FUNCTION_BLOCK FB_HMI_RP_BRANCH_A EXTENDS FB_HMI_COMPONENT
VAR_INPUT
END_VAR
VAR_OUTPUT
END_VAR
VAR
END_VAR

END_FUNCTION_BLOCK

(* stored: Version 1.1.0.1, ProductVersion 3.1.4024.14
   POU FB_HMI_RP_BRANCH_A: Id {5a11f014-8658-40c3-a394-553fde72265c}, SpecialFunc None *)
